TYPE Wsl15_RegSegmentXCfg :
STRUCT
	(*IO-link endian fuck zooi mother piieeeeeeeeeeeppppp*)	
	ManualSegmentWidth:BYTE;					//0
	ManualSegmentOffset:BYTE;					//0
	Direction:BYTE;								//0=up
	PercentWidthColor:BYTE;						//50
	ScrollBounceType:BYTE;						//0
	Color2Intensity:eWsl15_Intensity;
	Color2:eWsl15_Color;
	PulsePattern:BYTE;							//0=normal
	Speed:BYTE;									//0=medium,1=fast,2=slow,3=custom
	Color1Intensity:eWsl15_Intensity;
	Color1:eWsl15_Color;
	Animation:eWsl15_Animation;
	BasicFlashRate:BYTE;
	BasicColor:eWsl15_Color;
			
	(*beckhoff  endian
	BasicColor:eWsl15_Color;
	BasicFlashRate:BYTE;						//0=medium,1=fast,2=slow,3=custom
	Animation:eWsl15_Animation;
	Color1:eWsl15_Color;
	Color1Intensity:eWsl15_Intensity;
	Speed:BYTE;									//0=medium,1=fast,2=slow,3=custom
	PulsePattern:BYTE;							//0=normal
	Color2:eWsl15_Color;
	Color2Intensity:eWsl15_Intensity;
	ScrollBounceType:BYTE;						//0
	PercentWidthColor:BYTE;						//50
	Direction:BYTE;								//0=up
	ManualSegmentOffset:BYTE;					//0
	ManualSegmentWidth:BYTE;					//0
	*)
END_STRUCT
END_TYPE

(* stored: Version 1.1.0.1
   DUT Wsl15_RegSegmentXCfg: Id {180c4308-886a-47bd-8bac-769e2319c1ba} *)
